// Mitsubishi GX Works2 project: אוטומציה עבודה 2 עובד   PLC: FX3G

// global labels: Global1
VAR_GLOBAL
  on_off AT X010 : BOOL;
  light1 AT Y010 : BOOL;
  input1_kemach AT D1110 : REAL;
  input2_water AT D1120 : REAL;
  input3_shmarim AT D1130 : REAL;
  input4_oil AT D1140 : REAL;
  input5_tavlinim AT D1150 : REAL;
  kemach AT D1160 : REAL;
  water AT D1170 : REAL;
  shmarim AT D1180 : REAL;
  oil AT D1190 : REAL;
  tavlinim AT D1200 : REAL;
  enough_kemach AT M61 : BOOL;
  min_kemach AT E100 : REAL;
  enough_chala AT M60 : BOOL;
  enough_shmarim AT M62 : BOOL;
END_VAR
VAR_GLOBAL CONSTANT
  const2 : REAL := 2.0;
END_VAR
VAR_GLOBAL
  enough_water AT M63 : BOOL;
  enough_oil AT M64 : BOOL;
  emergency_stop AT X007 : BOOL;
  end_day_light AT M3 : BOOL;
END_VAR
VAR_GLOBAL CONSTANT
  const5 : REAL := 5;
  const03 : REAL := 0.3;
  const01 : REAL := 0.1;
END_VAR
VAR_GLOBAL
  enough_tavlinim AT M67 : BOOL;
  start_materials AT X002 : BOOL;
END_VAR
VAR_GLOBAL CONSTANT
  const30 : INT := 30;
  const_kemah_100 : REAL := 100;
  const_water_50 : REAL := 50;
  const_shmarim_20 : REAL := 20;
  const_shemen_30 : REAL := 30;
  const_tavlinim_10 : REAL := 10.0;
END_VAR
VAR_GLOBAL
  light05 AT Y005 : BOOL;
  lisha AT X001 : BOOL;
  stop_lisha AT M1 : BOOL;
  hatfaha AT X011 : BOOL;
  C0_HATFAHA AT CC0 : BOOL;
END_VAR
VAR_GLOBAL CONSTANT
  const_limit : INT := 2;
END_VAR
VAR_GLOBAL
  out_c0 AT CS0 : BOOL;
  light02 AT Y002 : BOOL;
END_VAR
VAR_GLOBAL CONSTANT
  count20 : INT := 5;
END_VAR
VAR_GLOBAL
  timer3 AT TC3 : BOOL;
  timer3_out AT TS3 : BOOL;
  light03 AT Y003 : BOOL;
  blink_start2 AT M95 : BOOL;
  light01 AT Y001 : BOOL;
  timer4 AT TC4 : BOOL;
  timer4_out AT TS4 : BOOL;
  timer5 AT TC5 : BOOL;
  timer5_out AT TS5 : BOOL;
  c2_blink_counter AT CC2 : BOOL;
END_VAR
VAR_GLOBAL CONSTANT
  const3sec : INT := 4;
END_VAR
VAR_GLOBAL
  counter2 AT CS2 : BOOL;
  start_afia AT M20 : BOOL;
  timer6 AT TC6 : BOOL;
  timer6_out AT TS6 : BOOL;
END_VAR
VAR_GLOBAL CONSTANT
  const40 : INT := 40;
END_VAR
VAR_GLOBAL
  light04 AT Y004 : BOOL;
  light06 AT Y006 : BOOL;
  light_fake AT M90 : BOOL;
  light_fake2 AT M91 : BOOL;
  new AT M23 : BOOL;
  counter10 AT CS10 : BOOL;
  timer10 AT TC10 : BOOL;
END_VAR
VAR_GLOBAL CONSTANT
  count100 : INT := 5;
END_VAR
VAR_GLOBAL
  timer10_out AT TS10 : BOOL;
  timer11 AT TC11 : BOOL;
  timer11_out AT TS11 : BOOL;
  light98 AT M98 : BOOL;
  blink_start10 AT M97 : BOOL;
  c10_blink_counter AT CC10 : BOOL;
END_VAR
VAR_GLOBAL CONSTANT
  const300 : INT := 4;
END_VAR
VAR_GLOBAL
  switch_QA AT X003 : BOOL;
  isMore AT M200 : BOOL;
  isLess AT M300 : BOOL;
END_VAR
VAR_GLOBAL CONSTANT
  add_kemach : REAL := 100;
END_VAR
VAR_GLOBAL
  michal_kemach AT D1300 : REAL;
END_VAR
VAR_GLOBAL CONSTANT
  add_water : REAL := 50;
END_VAR
VAR_GLOBAL
  michal_water AT D1310 : REAL;
END_VAR
VAR_GLOBAL CONSTANT
  add_shmarim : REAL := 20;
END_VAR
VAR_GLOBAL
  michal_shmarim AT D1320 : REAL;
END_VAR
VAR_GLOBAL CONSTANT
  add_oil : REAL := 30;
END_VAR
VAR_GLOBAL
  michal_oil AT D1330 : REAL;
END_VAR
VAR_GLOBAL CONSTANT
  add_tavlinim : REAL := 10;
END_VAR
VAR_GLOBAL
  michal_tavlinim AT D1340 : REAL;
  ta_hatfaca AT D1360 : REAL;
  tavnit AT D1370 : REAL;
END_VAR
VAR_GLOBAL CONSTANT
  reset : REAL;
  min_400 : INT := 400;
  max_2000 : INT := 2000;
END_VAR
VAR_GLOBAL
  timer13 AT TC13 : BOOL;
  const13 AT K50 : INT;
  madaf_chalot AT D1380 : REAL;
  M_108 AT M108 : BOOL;
  mixer AT D1400 : REAL;
  M_555 AT M495 : BOOL;
  M_494 AT M494 : BOOL;
  M_493 AT M493 : BOOL;
  good_chala2 AT M333 : BOOL;
  analog_input AT D8281 : INT;
  analog_output AT D8282 : INT;
  count_trying AT CC6 : BOOL;
  timer13_out AT TS13 : BOOL;
  cs6 AT CS6 : BOOL;
END_VAR
VAR_GLOBAL CONSTANT
  trying_to1 : INT := 3;
END_VAR
VAR_GLOBAL
  reset_newday AT M111 : BOOL;
  M_458 AT M458 : BOOL;
  M_321 AT M321 : BOOL;
  iteration AT M251 : BOOL;
END_VAR

// task Task_01 (event TRUE, interval 0, priority 31): POU_01

PROGRAM POU_01
(* structured ladder/FBD written out as ST: instructions are called as NAME(EN, inputs, outputs); _pN, _eN, _tN stand for wires *)
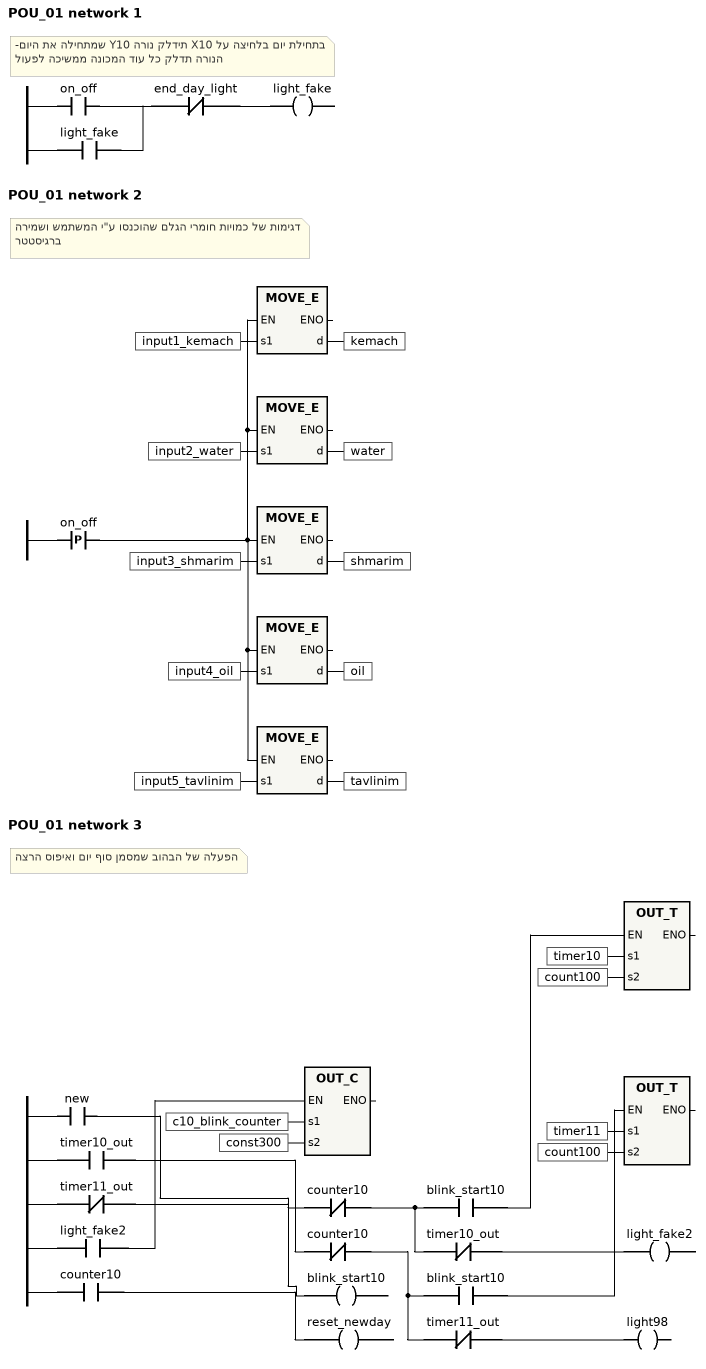
(* network 1 *)
(* בתחילת יום בלחיצה על X10 תידלק נורה Y10 שמתחילה את היום- הנורה תדלק כל עוד המכונה ממשיכה לפעול *)
light_fake := (on_off OR light_fake) AND NOT end_day_light;
(* network 2 *)
(* דגימות של כמויות חומרי הגלם שהוכנסו ע"י המשתמש ושמירה ברגיסטטר *)
_p1 := LDP(TRUE, on_off);
MOVE_E(_p1, input1_kemach, kemach);
MOVE_E(_p1, input2_water, water);
MOVE_E(_p1, input3_shmarim, shmarim);
MOVE_E(_p1, input4_oil, oil);
MOVE_E(_p1, input5_tavlinim, tavlinim);
(* network 3 *)
(* הפעלה של הבהוב שמסמן סוף יום ואיפוס הרצה *)
_p1 := new AND NOT counter10;
OUT_T(_p1 AND blink_start10, timer10, count100);
light_fake2 := _p1 AND NOT timer10_out;
_p2 := timer10_out AND NOT counter10;
OUT_T(_p2 AND blink_start10, timer11, count100);
light98 := _p2 AND NOT timer11_out;
blink_start10 := NOT timer11_out;
OUT_C(light_fake2, c10_blink_counter, const300);
reset_newday := counter10;
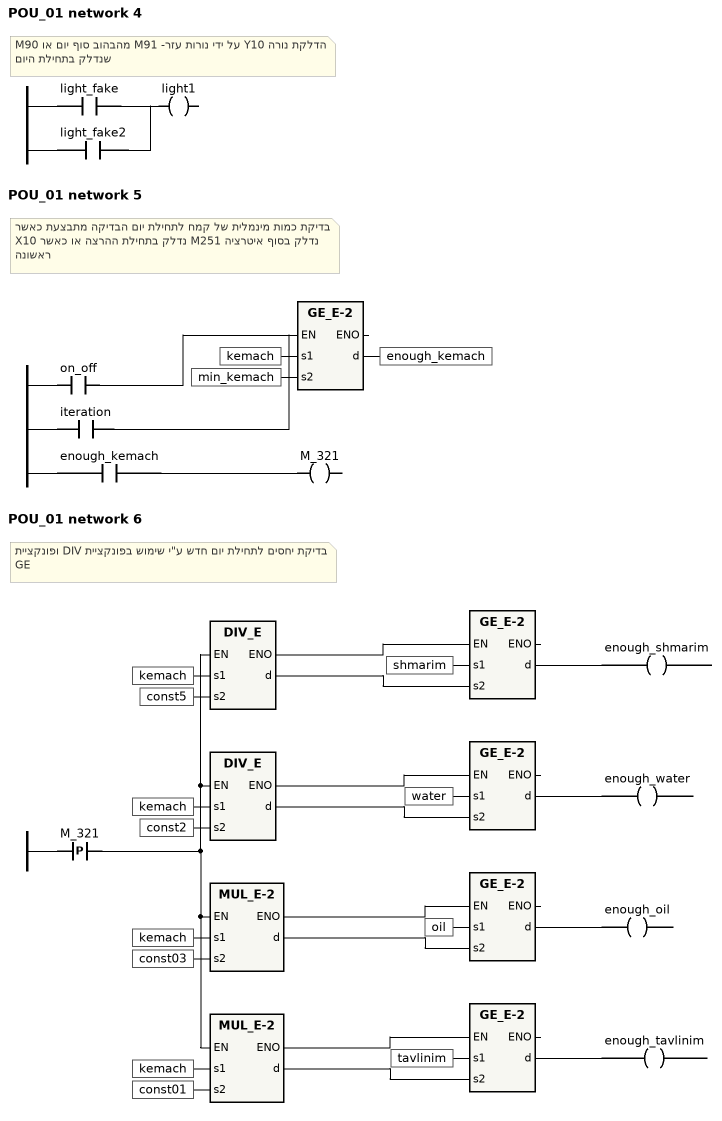
(* network 4 *)
(* הדלקת נורה Y10 על ידי נורות עזר- M91 מהבהוב סוף יום או M90 שנדלק בתחילת היום *)
light1 := light_fake OR light_fake2;
(* network 5 *)
(* בדיקת כמות מינמלית של קמח לתחילת יום הבדיקה מתבצעת כאשר X10 נדלק בתחילת ההרצה או כאשר M251 נדלק בסוף איטרציה ראשונה *)
GE_E(on_off OR iteration, kemach, min_kemach, enough_kemach);
M_321 := enough_kemach;
(* network 6 *)
(* בדיקת יחסים לתחילת יום חדש ע"י שימוש בפונקציית DIV ופונקציית GE *)
_p1 := LDP(TRUE, M_321);
_e3 := DIV_E(_p1, kemach, const5, _t2);
GE_E(_e3, shmarim, _t2, _t4);
enough_shmarim := _t4;
_e6 := DIV_E(_p1, kemach, const2, _t5);
GE_E(_e6, water, _t5, _t7);
enough_water := _t7;
_e9 := MUL_E(_p1, kemach, const03, _t8);
GE_E(_e9, oil, _t8, _t10);
enough_oil := _t10;
_e12 := MUL_E(_p1, kemach, const01, _t11);
GE_E(_e12, tavlinim, _t11, _t13);
enough_tavlinim := _t13;
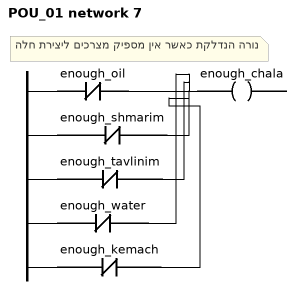
(* network 7 *)
(* נורה הנדלקת כאשר אין מספיק מצרכים ליצירת חלה *)
enough_chala := (NOT enough_oil) OR (NOT enough_shmarim) OR (NOT enough_tavlinim) OR (NOT enough_water) OR (NOT enough_kemach);
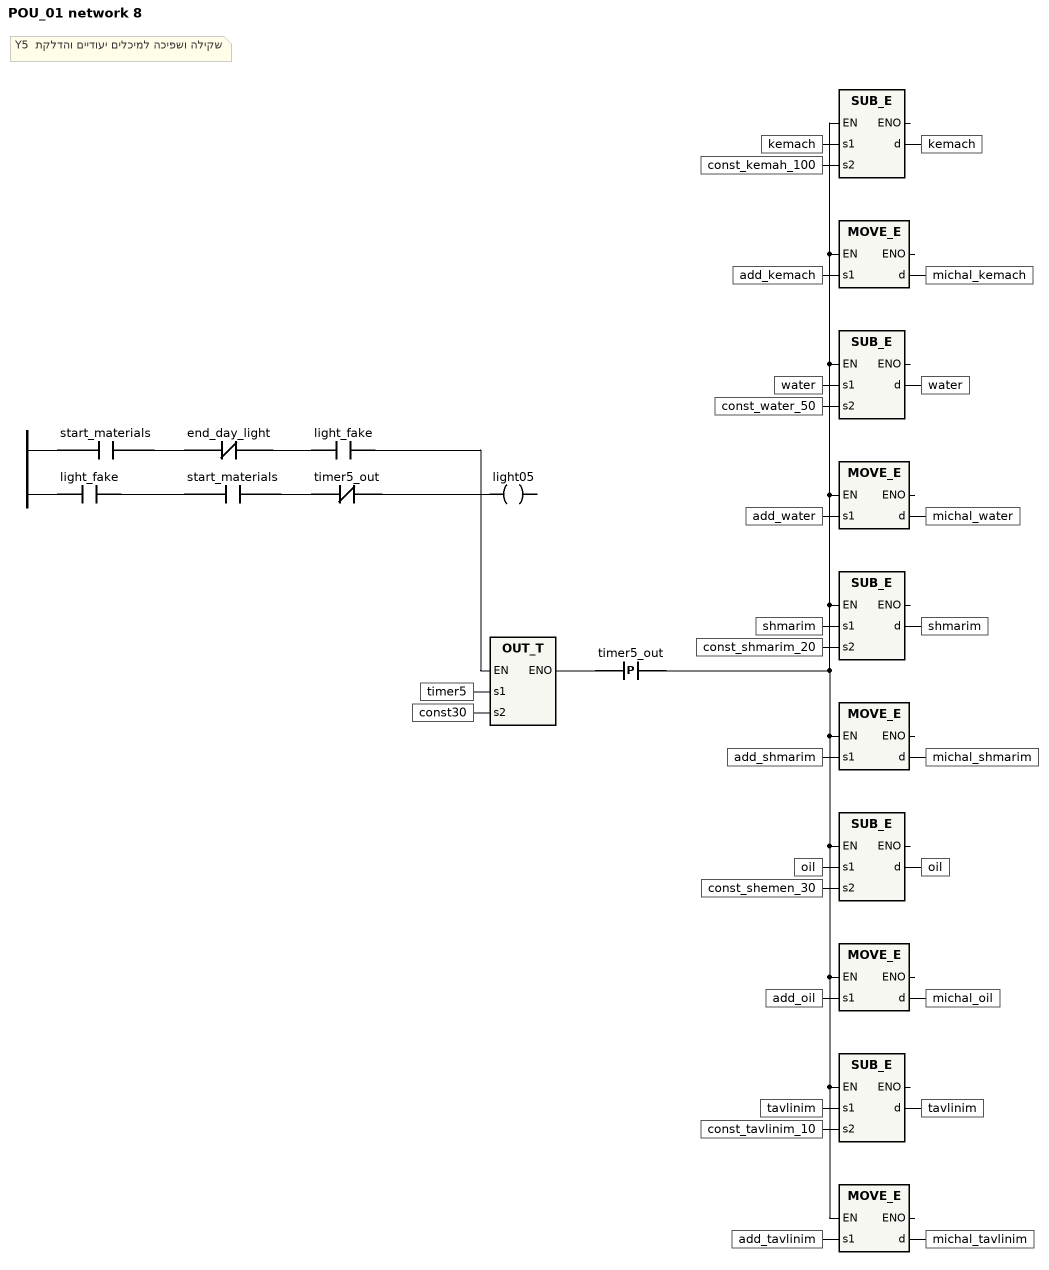
(* network 8 *)
(* שקילה ושפיכה למיכלים יעודיים והדלקת  Y5 *)
_e1 := OUT_T(start_materials AND NOT end_day_light AND light_fake, timer5, const30);
_p2 := _e1 AND LDP(TRUE, timer5_out);
SUB_E(_p2, kemach, const_kemah_100, kemach);
MOVE_E(_p2, add_kemach, michal_kemach);
light05 := light_fake AND start_materials AND NOT timer5_out;
SUB_E(_p2, water, const_water_50, water);
MOVE_E(_p2, add_water, michal_water);
SUB_E(_p2, shmarim, const_shmarim_20, shmarim);
MOVE_E(_p2, add_shmarim, michal_shmarim);
SUB_E(_p2, oil, const_shemen_30, oil);
MOVE_E(_p2, add_oil, michal_oil);
SUB_E(_p2, tavlinim, const_tavlinim_10, tavlinim);
MOVE_E(_p2, add_tavlinim, michal_tavlinim);
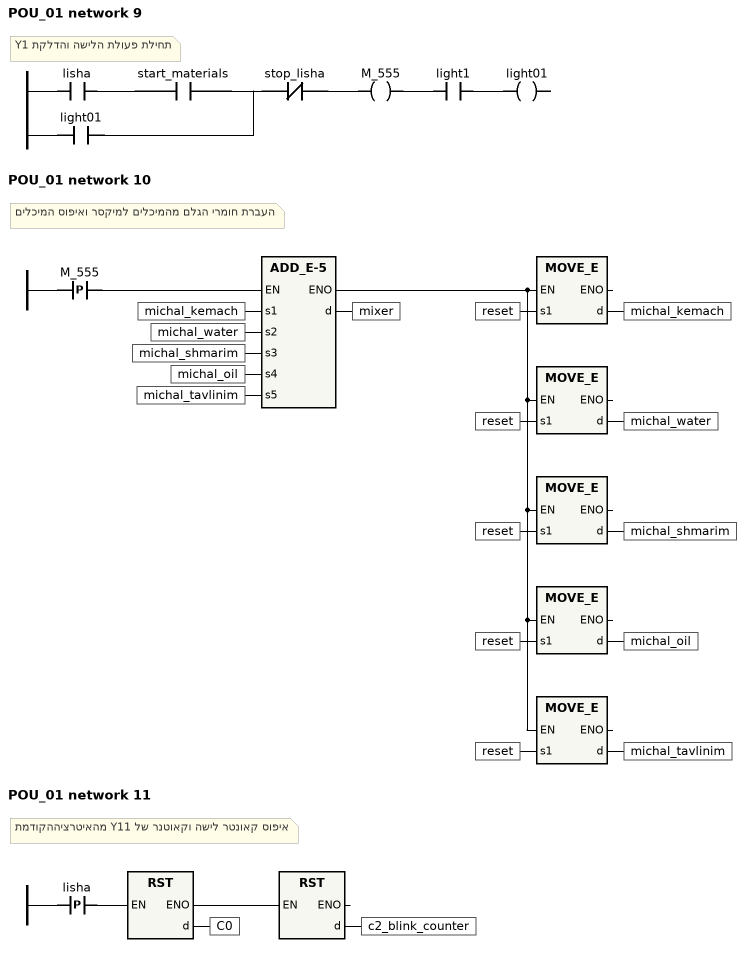
(* network 9 *)
(* תחילת פעולת הלישה והדלקת Y1 *)
_p1 := ((lisha AND start_materials) OR light01) AND NOT stop_lisha;
M_555 := _p1;
light01 := _p1 AND light1;
(* network 10 *)
(* העברת חומרי הגלם מהמיכלים למיקסר ואיפוס המיכלים *)
_e1 := ADD_E(LDP(TRUE, M_555), michal_kemach, michal_water, michal_shmarim, michal_oil, michal_tavlinim, mixer);
MOVE_E(_e1, reset, michal_kemach);
MOVE_E(_e1, reset, michal_water);
MOVE_E(_e1, reset, michal_shmarim);
MOVE_E(_e1, reset, michal_oil);
MOVE_E(_e1, reset, michal_tavlinim);
(* network 11 *)
(* איפוס קאונטר לישה וקאוטנר של Y11 מהאיטרציההקודמת *)
_e1 := RST(LDP(TRUE, lisha), C0);
RST(_e1, c2_blink_counter);
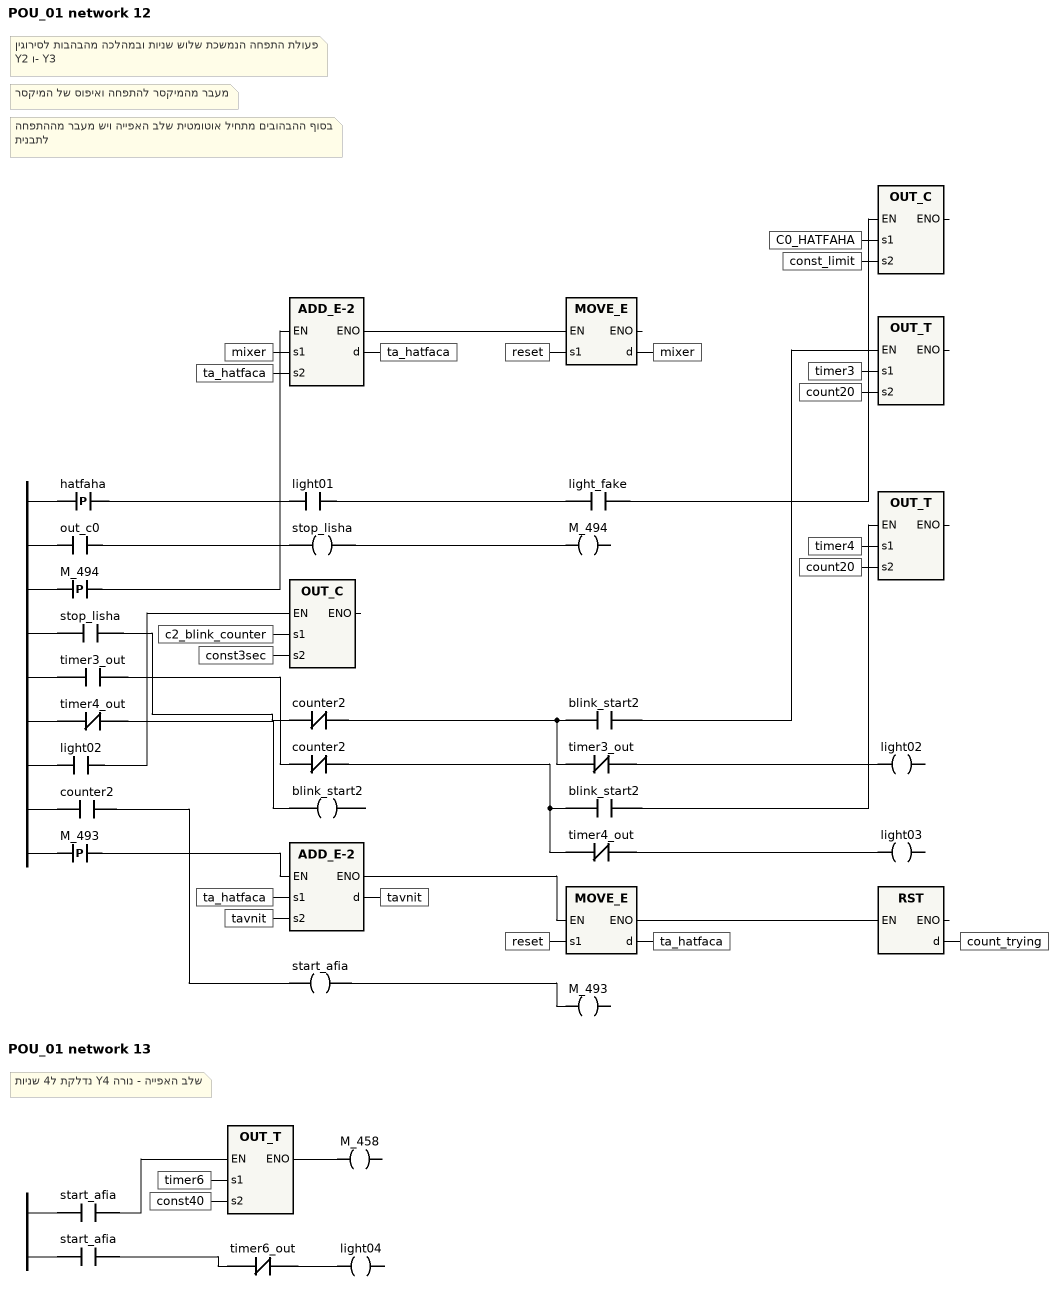
(* network 12 *)
(* פעולת התפחה הנמשכת שלוש שניות ובמהלכה מהבהבות לסירוגין Y2 ו- Y3 *)
(* מעבר מהמיקסר להתפחה ואיפוס של המיקסר *)
(* בסוף ההבהובים מתחיל אוטומטית שלב האפייה ויש מעבר מההתפחה לתבנית *)
OUT_C(LDP(TRUE, hatfaha) AND light01 AND light_fake, C0_HATFAHA, const_limit);
stop_lisha := out_c0;
M_494 := out_c0;
_e1 := ADD_E(LDP(TRUE, M_494), mixer, ta_hatfaca, ta_hatfaca);
MOVE_E(_e1, reset, mixer);
_p2 := stop_lisha AND NOT counter2;
OUT_T(_p2 AND blink_start2, timer3, count20);
light02 := _p2 AND NOT timer3_out;
_p3 := timer3_out AND NOT counter2;
OUT_T(_p3 AND blink_start2, timer4, count20);
light03 := _p3 AND NOT timer4_out;
blink_start2 := NOT timer4_out;
OUT_C(light02, c2_blink_counter, const3sec);
start_afia := counter2;
M_493 := counter2;
_e4 := ADD_E(LDP(TRUE, M_493), ta_hatfaca, tavnit, tavnit);
_e5 := MOVE_E(_e4, reset, ta_hatfaca);
RST(_e5, count_trying);
(* network 13 *)
(* שלב האפייה - נורה Y4 נדלקת ל4 שניות *)
_e1 := OUT_T(start_afia, timer6, const40);
M_458 := _e1;
light04 := start_afia AND NOT timer6_out;
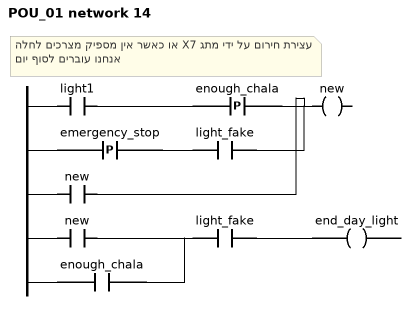
(* network 14 *)
(* עצירת חירום על ידי מתג X7 או כאשר אין מספיק מצרכים לחלה אנחנו עוברים לסוף יום *)
new := (light1 AND LDP(TRUE, enough_chala)) OR (LDP(TRUE, emergency_stop) AND light_fake) OR new;
end_day_light := (new OR enough_chala) AND light_fake;
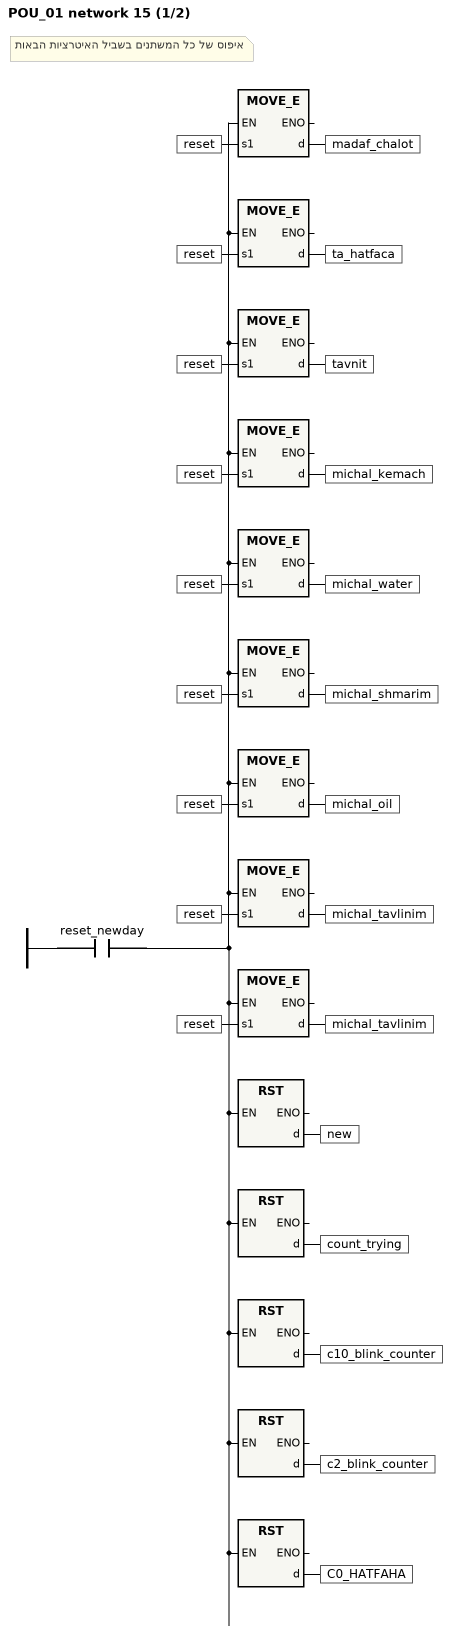
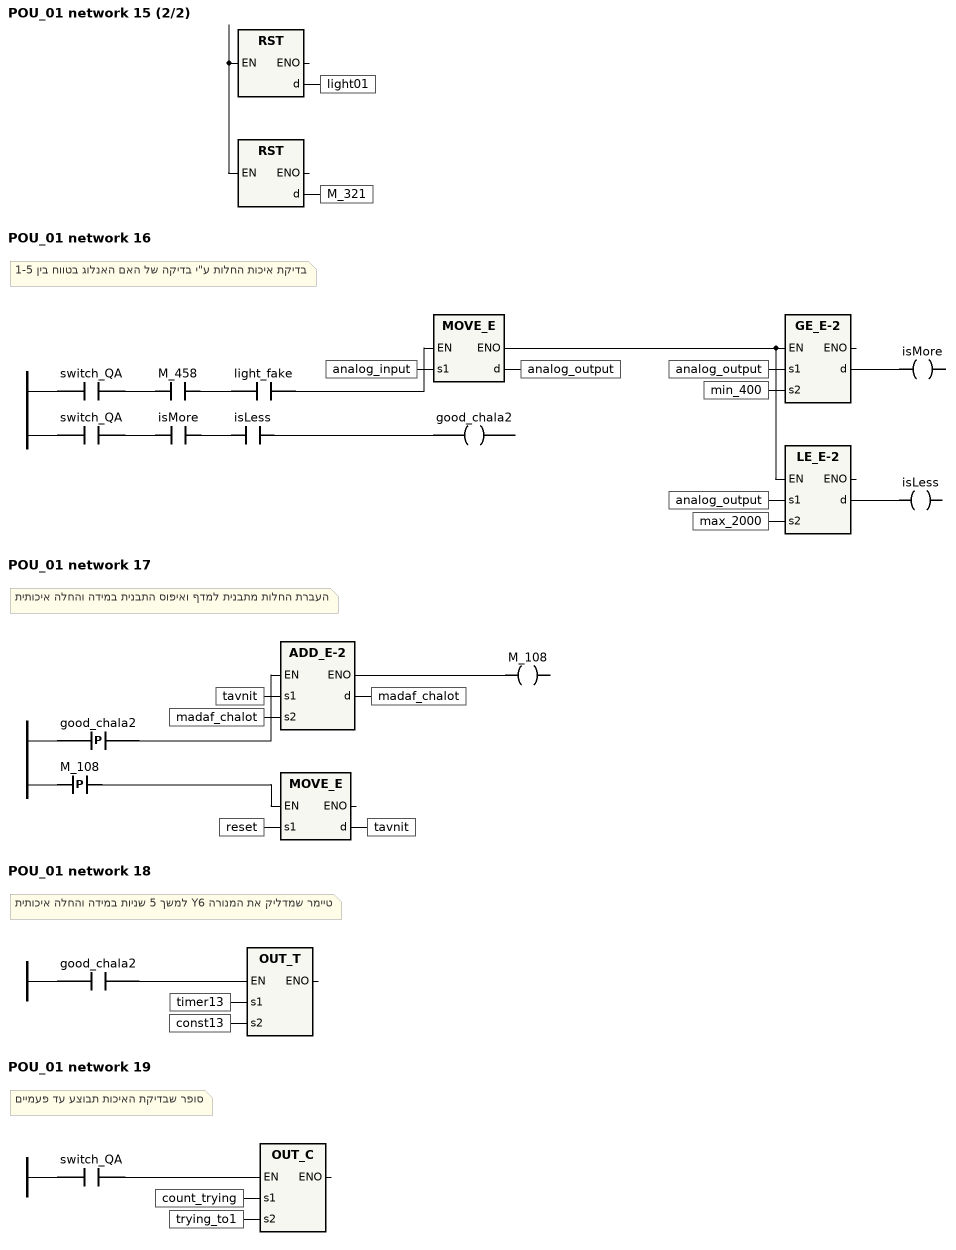
(* network 15 *)
(* איפוס של כל המשתנים בשביל האיטרציות הבאות *)
MOVE_E(reset_newday, reset, madaf_chalot);
MOVE_E(reset_newday, reset, ta_hatfaca);
MOVE_E(reset_newday, reset, tavnit);
MOVE_E(reset_newday, reset, michal_kemach);
MOVE_E(reset_newday, reset, michal_water);
MOVE_E(reset_newday, reset, michal_shmarim);
MOVE_E(reset_newday, reset, michal_oil);
MOVE_E(reset_newday, reset, michal_tavlinim);
MOVE_E(reset_newday, reset, michal_tavlinim);
RST(reset_newday, new);
RST(reset_newday, count_trying);
RST(reset_newday, c10_blink_counter);
RST(reset_newday, c2_blink_counter);
RST(reset_newday, C0_HATFAHA);
RST(reset_newday, light01);
RST(reset_newday, M_321);
(* network 16 *)
(* בדיקת איכות החלות ע"י בדיקה של האם האנלוג בטווח בין 1-5 *)
_e1 := MOVE_E(switch_QA AND M_458 AND light_fake, analog_input, analog_output);
GE_E(_e1, analog_output, min_400, _t2);
isMore := _t2;
LE_E(_e1, analog_output, max_2000, _t3);
isLess := _t3;
good_chala2 := switch_QA AND isMore AND isLess;
(* network 17 *)
(* העברת החלות מתבנית למדף ואיפוס התבנית במידה והחלה איכותית *)
_e1 := ADD_E(LDP(TRUE, good_chala2), tavnit, madaf_chalot, madaf_chalot);
M_108 := _e1;
MOVE_E(LDP(TRUE, M_108), reset, tavnit);
(* network 18 *)
(* טיימר שמדליק את המנורה Y6 למשך 5 שניות במידה והחלה איכותית *)
OUT_T(good_chala2, timer13, const13);
(* network 19 *)
(* סופר שבדיקת האיכות תבוצע עד פעמיים *)
OUT_C(switch_QA, count_trying, trying_to1);
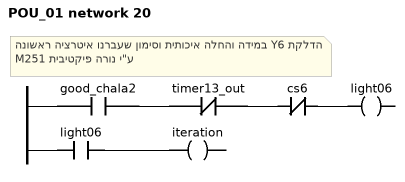
(* network 20 *)
(* הדלקת Y6 במידה והחלה איכותית וסימון שעברנו איטרציה ראשונה ע"י נורה פיקטיבית M251 *)
light06 := good_chala2 AND NOT timer13_out AND NOT cs6;
iteration := light06;
END_PROGRAM
